PROGRAM JIG_GRAB
VAR
END_VAR

END_PROGRAM

(* stored: Version 1.1.0.1, ProductVersion 3.1.4022.18
   POU JIG_GRAB: Id {0b02a691-20a2-49ff-85ea-fb6d489239c2}, SpecialFunc None *)
